FUNCTION GearType : STRING[80]
VAR_INPUT
	nGearType	:	BYTE;
END_VAR
VAR
	i: INT;
	aText	:	ARRAY [0..7] OF STRING[80];
END_VAR

GearType := '';
	aText[0] := 'Output is an electronic switch';
	aText[1] := 'Output is a relay with default open contacts';
	aText[2] := 'Output is a relay with default closed contacts';
	aText[3] := 'Output has a transient suppressor';
	aText[4] := 'Load inrush current limitation is integrated';
	aText[5] := '';
	aText[6] := '';
	aText[7] := '';
FOR i := 0 TO 7 DO
	IF nGearType.0 THEN
		GearType := aText[i];
	ELSE
		GearType := '';
	END_IF
	nGearType := ROR (nGearType,1);
END_FOR

IF (nGearType.1 AND nGearType.2)	THEN 
	GearType := 'Latched Output, the latched state does not change when power is removed';
END_IF

END_FUNCTION

(* stored: Version 1.1.0.1, ProductVersion 3.1.4024.12
   POU GearType: Id {7c05af54-4669-4e6f-aff0-b04a6bb76b79}, SpecialFunc None *)
